{attribute 'qualified_only'}
{attribute 'strict'}
TYPE TIoKind :
(
	DigitalIn := 0, DigitalOut, AnalogIn, AnalogOut
);
END_TYPE

(* stored: Version 1.1.0.1, ProductVersion 3.1.4024.3
   DUT TIoKind: Id {2219ce45-118e-4c6a-a822-5e09aa3196d1} *)
